// TIA Portal V20 export
FUNCTION_BLOCK "FB_DigitalInputs"   // FB210, SCL
{ S7_Optimized_Access := 'TRUE' }
// stored: AutoNumber false, MemoryReserve 100, SetENOAutomatically false
   VAR
      sFreeI0_0 : "FB_DigitalInput";
      sX_AxisBrakePressCtrl : "FB_DigitalInput";
      sY_AxisBrakePressCtrl : "FB_DigitalInput";
      sBreakerCtrl : "FB_DigitalInput";
      sCabinetTemperatureCtrl : "FB_DigitalInput";
      sUPS_PowerFailure : "FB_DigitalInput";
      sAirPressureCtrl : "FB_DigitalInput";
      sShutterClosed : "FB_DigitalInput";
      sAirDryerOK : "FB_DigitalInput";
      sUPS_BatteryOK : "FB_DigitalInput";
      sFrontDoorClosed : "FB_DigitalInput";
      sInfeedReadyOK_Start : "FB_DigitalInput";
      sCoolingOK : "FB_DigitalInput";
      sFreeI1_5 : "FB_DigitalInput";
      sPowerReady : "FB_DigitalInput";
      sAlarmI2T : "FB_DigitalInput";
      sHeadLaserBusy : "FB_DigitalInput";
      sHeadLaserBreaker { S7_SetPoint := 'True'} : "FB_DigitalInput";
      sFrontDoorLocked { S7_SetPoint := 'True'} : "FB_DigitalInput";
      sUPS_CommonAlarm { S7_SetPoint := 'True'} : "FB_DigitalInput";
      sUPS_BatteryLow { S7_SetPoint := 'True'} : "FB_DigitalInput";
      sFreeI2_5 { S7_SetPoint := 'True'} : "FB_DigitalInput";
      sHeadChillerHighPressure { S7_SetPoint := 'True'} : "FB_DigitalInput";
      sHeadChillerWaterTemperature { S7_SetPoint := 'True'} : "FB_DigitalInput";
      sHeadChillerFlow { S7_SetPoint := 'True'} : "FB_DigitalInput";
      sHeadChillerCollectivFault { S7_SetPoint := 'True'} : "FB_DigitalInput";
      sHeadChillerWaterLevel { S7_SetPoint := 'True'} : "FB_DigitalInput";
      sUPS_ByPassActive { S7_SetPoint := 'True'} : "FB_DigitalInput";
      sHeadChillerAmbiantTemperature { S7_SetPoint := 'True'} : "FB_DigitalInput";
      sFreeI3_5 { S7_SetPoint := 'True'} : "FB_DigitalInput";
      sFreeI3_6 { S7_SetPoint := 'True'} : "FB_DigitalInput";
      sFreeI3_7 { S7_SetPoint := 'True'} : "FB_DigitalInput";
      sLoadClampOpened { S7_SetPoint := 'True'} : "FB_DigitalInput";
      sLoadClampNotClosedWithPart { S7_SetPoint := 'True'} : "FB_DigitalInput";
      sUnloadClampOpened { S7_SetPoint := 'True'} : "FB_DigitalInput";
      sUPS_Fault { S7_SetPoint := 'True'} : "FB_DigitalInput";
      sInternalGateLocked { S7_SetPoint := 'True'} : "FB_DigitalInput";
      sExternalGateLocked { S7_SetPoint := 'True'} : "FB_DigitalInput";
      sInverterActive { S7_SetPoint := 'True'} : "FB_DigitalInput";
      sUnloadClampNotClosedWithPart { S7_SetPoint := 'True'} : "FB_DigitalInput";
      sFreeI5_0 { S7_SetPoint := 'True'} : "FB_DigitalInput";
      sFreeI5_1 { S7_SetPoint := 'True'} : "FB_DigitalInput";
      sInternalGateOpened { S7_SetPoint := 'True'} : "FB_DigitalInput";
      sExternalGateOpened { S7_SetPoint := 'True'} : "FB_DigitalInput";
      sPowerMeterBackCtrl { S7_SetPoint := 'True'} : "FB_DigitalInput";
      sPowerMeterFrontCtrl { S7_SetPoint := 'True'} : "FB_DigitalInput";
      sFreeI5_6 { S7_SetPoint := 'True'} : "FB_DigitalInput";
      sFreeI5_7 { S7_SetPoint := 'True'} : "FB_DigitalInput";
      sHeadChillerCutOff { S7_SetPoint := 'True'} : "FB_DigitalInput";
      sHeadChillerTemperature { S7_SetPoint := 'True'} : "FB_DigitalInput";
      sFreeI6_2 { S7_SetPoint := 'True'} : "FB_DigitalInput";
      sFreeI6_3 { S7_SetPoint := 'True'} : "FB_DigitalInput";
      sClampingOpenCtrl { S7_SetPoint := 'True'} : "FB_DigitalInput";
      sB_Axis_BrakeReleasedCtrl { S7_SetPoint := 'True'} : "FB_DigitalInput";
      sFreeI6_6 { S7_SetPoint := 'True'} : "FB_DigitalInput";
      sB_AxisReferencePoint { S7_SetPoint := 'True'} : "FB_DigitalInput";
      sSourceChillerHighPressure { S7_SetPoint := 'True'} : "FB_DigitalInput";
      sSourceChillerWaterTemperature { S7_SetPoint := 'True'} : "FB_DigitalInput";
      sSourceChillerFlow { S7_SetPoint := 'True'} : "FB_DigitalInput";
      sSourceChillerCollectivFault { S7_SetPoint := 'True'} : "FB_DigitalInput";
      sSourceChillerWaterLevel { S7_SetPoint := 'True'} : "FB_DigitalInput";
      sSourceChillerAmbiantTemperature { S7_SetPoint := 'True'} : "FB_DigitalInput";
      sSourceChillerCutOff { S7_SetPoint := 'True'} : "FB_DigitalInput";
      sSourceChillerTemperature { S7_SetPoint := 'True'} : "FB_DigitalInput";
   END_VAR
BEGIN
   REGION Description head
       //==================================================================================
       // POSALUX Swiss SA / (C) Copyright 2025
       //----------------------------------------------------------------------------------
       // Title: Digital Inputs mapping
       // Comment/Function: Digital Inputs mapping
       // Author: Fabien WALDT
       // Engineering: TIA Portal v17
       //----------------------------------------------------------------------------------
       // Change log table:
       // Version  | Date     | Expert in charge | Changes applied
       // ---------|----------|------------------|-----------------------------------------
       // 00.00.01 | 20250423 | WFA              | First released version
       // =================================================================================
   END_REGION

       // ET200SP Mapping
   REGION I0.0 - I1.7 : DI 16x24VDC ST Slot 1
       #sFreeI0_0(iHWStatus := "DI_FreeI0_0");
       #sX_AxisBrakePressCtrl(iHWStatus := "DI_X_AxisBrakePressCtrl");
       #sY_AxisBrakePressCtrl(iHWStatus := "DI_Y_AxisBrakePressCtrl");
       #sBreakerCtrl(iHWStatus := "DI_BreakerCtrl");
       #sCabinetTemperatureCtrl(iHWStatus := "DI_CabinetTemperatureCtrl");
       #sUPS_PowerFailure(iHWStatus := "DI_UPS_PowerFailure");
       #sAirPressureCtrl(iHWStatus := "DI_AirPressureCtrl");
       #sShutterClosed(iHWStatus := "DI_ShutterClosed");
       //
       #sAirDryerOK(iHWStatus := "DI_AirDryerOK");
       #sUPS_BatteryOK(iHWStatus := "DI_UPS_BatteryOK");
       #sFrontDoorClosed(iHWStatus := "DI_FrontDoorClosed");
       #sInfeedReadyOK_Start(iHWStatus := "DI_InfeedReadyOK_Start");
       #sCoolingOK(iHWStatus := "DI_CoolingOK");
       #sFreeI1_5(iHWStatus := "DI_FreeI1_5");
       #sPowerReady(iHWStatus := "DI_PowerReady");
       #sAlarmI2T(iHWStatus := "DI_AlarmI2T");
   END_REGION

   REGION I2.0 - I3.7 : DI 16x24VDC ST Slot 2
       #sHeadLaserBusy(iHWStatus := "DI_HeadLaserBusy");
       #sHeadLaserBreaker(iHWStatus := "DI_HeadLaserBreaker");
       #sFrontDoorLocked(iHWStatus := "DI_FrontDoorLocked");
       #sUPS_CommonAlarm(iHWStatus := "DI_UPS_CommonAlarm");
       #sUPS_BatteryLow(iHWStatus := "DI_UPS_BatteryLow");
       #sFreeI2_5(iHWStatus := "DI_FreeI2_5");
       #sHeadChillerHighPressure(iHWStatus := "DI_HeadChillerHighPressure");
       #sHeadChillerWaterTemperature(iHWStatus := "DI_HeadChillerWaterTemperature");
       //
       #sHeadChillerFlow(iHWStatus := "DI_HeadChillerFlow");
       #sHeadChillerCollectivFault(iHWStatus := "DI_HeadChillerCollectivFault");
       #sHeadChillerWaterLevel(iHWStatus := "DI_HeadChillerWaterLevel");
       #sUPS_ByPassActive(iHWStatus := "DI_UPSByPassActive");
       #sHeadChillerAmbiantTemperature(iHWStatus := "DI_HeadChillerAmbiantTemperature");
       #sFreeI3_5(iHWStatus := "DI_FreeI3_5");
       #sFreeI3_6(iHWStatus := "DI_FreeI3_6");
       #sFreeI3_7(iHWStatus := "DI_FreeI3_7");
   END_REGION

   REGION I4.0 - I5.7 : DI 16x24VDC ST Slot 3
       #sLoadClampOpened(iHWStatus := "DI_LoadClampOpened");
       #sLoadClampNotClosedWithPart(iHWStatus := "DI_LoadClampNotClosedWithPart");
       #sUnloadClampOpened(iHWStatus := "DI_UnloadClampOpened");
       #sUPS_Fault(iHWStatus := "DI_UPS_Fault");
       #sInternalGateLocked(iHWStatus := NOT "DI_InternalGateLocked");
       #sExternalGateLocked(iHWStatus := NOT "DI_ExternalGateLocked");
       #sInverterActive(iHWStatus := "DI_InverterActive");
       #sUnloadClampNotClosedWithPart(iHWStatus := "DI_UnloadClampNotClosedWithPart");
       //
       #sFreeI5_0(iHWStatus := "DI_FreeI5_0");
       #sFreeI5_1(iHWStatus := "DI_FreeI5_1");
       #sInternalGateOpened(iHWStatus := "DI_InternalGateOpened");
       #sExternalGateOpened(iHWStatus := "DI_ExternalGateOpened");
       #sPowerMeterBackCtrl(iHWStatus := "DI_PowerMeterBackCtrl");
       #sPowerMeterFrontCtrl(iHWStatus := "DI_PowerMeterFrontCtrl");
       #sFreeI5_6(iHWStatus := "DI_FreeI5_6");
       #sFreeI5_7(iHWStatus := "DI_FreeI5_7");
   END_REGION

   REGION I6.0 - I7.7 : DI 16x24VDC ST Slot 4
       #sHeadChillerCutOff(iHWStatus := "DI_HeadChillerCutOff");
       #sHeadChillerTemperature(iHWStatus := "DI_HeadChillerTemperature");
       #sFreeI6_2(iHWStatus := "DI_FreeI6_2");
       #sFreeI6_3(iHWStatus := "DI_FreeI6_3");
       #sClampingOpenCtrl(iHWStatus := "DI_ClampingOpenCtrl");
       #sB_Axis_BrakeReleasedCtrl(iHWStatus := "DI_B_AxisBrakeReleasedCtrl");
       #sFreeI6_6(iHWStatus := "DI_FreeI6.6");
       #sB_AxisReferencePoint(iHWStatus := "DI_B_AxisReferencePoint");
       //
       #sSourceChillerHighPressure(iHWStatus := "DI_SourceChillerHighPressure");
       #sSourceChillerWaterTemperature(iHWStatus := "DI_SourceChillerWaterTemperature");
       #sSourceChillerFlow(iHWStatus := "DI_SourceChillerFlow");
       #sSourceChillerCollectivFault(iHWStatus := "DI_SourceChillerCollectivFault");
       #sSourceChillerWaterLevel(iHWStatus := "DI_SourceChillerWaterLevel");
       #sSourceChillerAmbiantTemperature(iHWStatus := "DI_SourceChillerAmbiantTemperature");
       #sSourceChillerCutOff(iHWStatus := "DI_SourceChillerCutOff");
       #sSourceChillerTemperature(iHWStatus := "DI_SourceChillerTemperature");
   END_REGION
END_FUNCTION_BLOCK
